PROGRAM PRG_LARS_03_AddtitionalConvCtrl
VAR
	fbAddtitionalConvDelay	 : FB_TOFR;
END_VAR

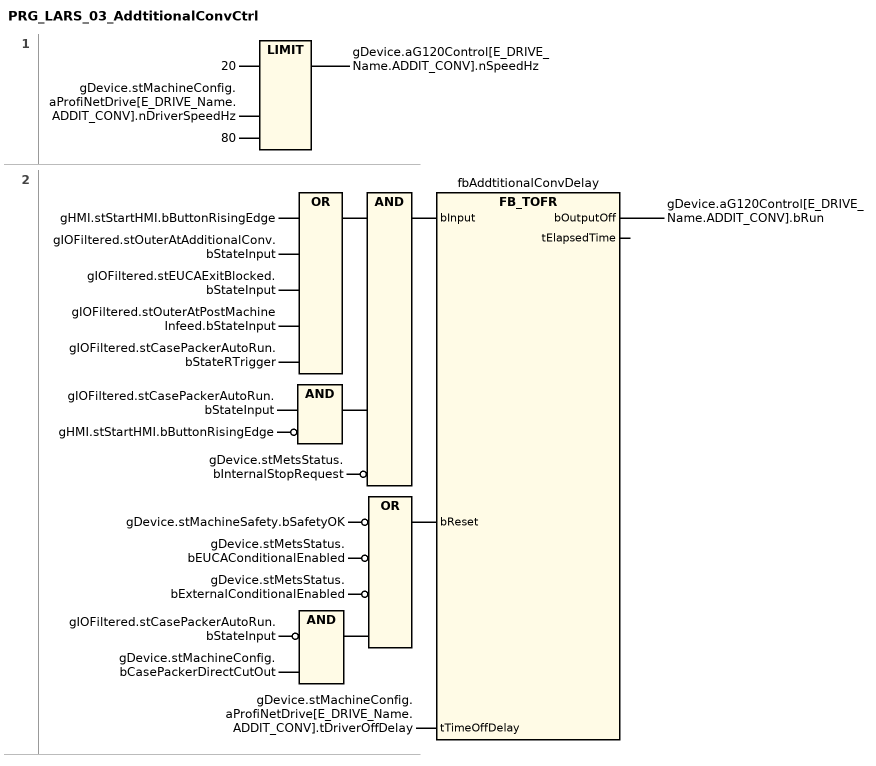
// NETWORK 1
gDevice.aG120Control[E_DRIVE_Name.ADDIT_CONV].nSpeedHz := LIMIT(20, gDevice.stMachineConfig.aProfiNetDrive[E_DRIVE_Name.ADDIT_CONV].nDriverSpeedHz, 80);

// NETWORK 2
fbAddtitionalConvDelay(
    bInput := (gHMI.stStartHMI.bButtonRisingEdge OR gIOFiltered.stOuterAtAdditionalConv.bStateInput OR gIOFiltered.stEUCAExitBlocked.bStateInput OR gIOFiltered.stOuterAtPostMachineInfeed.bStateInput OR gIOFiltered.stCasePackerAutoRun.bStateRTrigger) AND (gIOFiltered.stCasePackerAutoRun.bStateInput AND NOT gHMI.stStartHMI.bButtonRisingEdge) AND NOT gDevice.stMetsStatus.bInternalStopRequest,
    bReset := NOT gDevice.stMachineSafety.bSafetyOK OR NOT gDevice.stMetsStatus.bEUCAConditionalEnabled OR NOT gDevice.stMetsStatus.bExternalConditionalEnabled OR NOT gIOFiltered.stCasePackerAutoRun.bStateInput AND gDevice.stMachineConfig.bCasePackerDirectCutOut,
    tTimeOffDelay := gDevice.stMachineConfig.aProfiNetDrive[E_DRIVE_Name.ADDIT_CONV].tDriverOffDelay); // FB_TOFR
gDevice.aG120Control[E_DRIVE_Name.ADDIT_CONV].bRun := fbAddtitionalConvDelay.bOutputOff;

END_PROGRAM

(* stored: Version 1.1.0.1
   POU PRG_LARS_03_AddtitionalConvCtrl: Id {9aecfd48-038c-412c-9641-b2e088c4dae4}, SpecialFunc None *)
